{attribute 'hide'}
TYPE ST_Hidden :
STRUCT
    nX : INT;
END_STRUCT
END_TYPE

(* stored: Version 1.1.0.1
   DUT ST_Hidden: Id {55555555-5555-5555-5555-555555555505} *)
